// TIA Portal V19 export
DATA_BLOCK "A01_DEBUG"   // DB129
// stored: MemoryReserve 100
   VAR
      Force_Sinamics_CtrlSafe : Bool;
      Forse_Contactors_CtrlSafe : Bool;
      CoilHandling_Simulation : Struct
         Enable : Bool;
         S_StraightenerEntry : Bool;
         S_StraightenerExit : Bool;
         S_JBPinchExit : Bool;
         S_Downstream_Entry : Bool;
         LoopCtrl_Enable_FWD : Bool;
         LoopCtrl_Enable_BWD : Bool;
         LoopCtrl_SpeedOverride : LReal;
         Material_FWD_Velocity : LReal;
         Pb : Struct
            Enable : Bool;
            Fwd_MaterialFeed : Bool;
            Bwd_MaterialFeed : Bool;
            Fwd_Decoiler_Snubber : Bool;
            Bwd_Decoiler_Snubber : Bool;
            Fwd_Decoiler_Straight : Bool;
            Bwd_Decoiler_Straight : Bool;
            Fwd_Decoiler_Straight_Snubber : Bool;
            Bwd_Decoiler_Straight_Snubber : Bool;
         END_STRUCT;
         DecoilerInLine_Sensors : Struct
            Enable : Bool;
            Phc_Min : Bool;
            Phc_Max : Bool;
            Phc_SpeedAdjust : Bool;
         END_STRUCT;
         WeldDone : Bool;
         CutDone : Bool;
      END_STRUCT;
   END_VAR
BEGIN
END_DATA_BLOCK
